FUNCTION_BLOCK TIMER_TON3 (* Composite Function Block Type *)
  (* Standard: 61499-2 *)
  (* Version 0.0, 7/6/2016, gulzha, nxtControl GmbH, template *)
  PACKAGE Main;
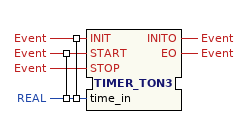
  EVENT_INPUT
    INIT WITH time_in; (* Initialization Request *)
    START WITH time_in; (* Normal Execution Request *)
    STOP;
  END_EVENT
  EVENT_OUTPUT
    INITO; (* Initialization Confirm *)
    EO; (* Delayed Event *)
  END_EVENT
  VAR_INPUT
    time_in : REAL;
  END_VAR
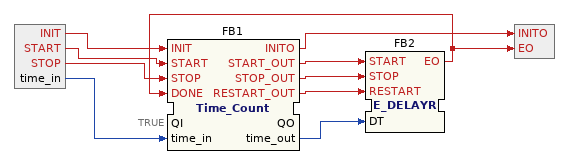
  FBS
    FB2 : E_DELAYR;
    FB1 : Time_Count(QI := TRUE);
  END_FBS
  EVENT_CONNECTIONS
    FB1.INITO TO INITO;
    INIT TO FB1.INIT;
    START TO FB1.START;
    STOP TO FB1.STOP;
    FB1.START_OUT TO FB2.START;
    FB1.STOP_OUT TO FB2.STOP;
    FB2.EO TO FB1.DONE;
    FB1.RESTART_OUT TO FB2.RESTART;
    FB2.EO TO EO;
  END_CONNECTIONS
  DATA_CONNECTIONS
    FB1.time_out TO FB2.DT;
    time_in TO FB1.time_in;
  END_CONNECTIONS
END_FUNCTION_BLOCK
